Staubli VAL3: Place.pgx

program Place(pointRx pPos)
begin
  movel(appro(pPos,{0,0,-50,0,0,0}),tTool1,mNomSpeed)
  delay(3)
  movel(appro(pPos,{0,0,-1,0,0,0}),tTool1,mSlow)
  delay(3)
  open(tTool1)
  movel(appro(pPos,{0,0,-50,0,0,0}),tTool1,mSlow)
  delay(3)
  close(tTool1)
end
